PROGRAM Pellet_Calibration
VAR
	SET_CALIBRATON_VALUE : BOOL;

	
	
	Pellet_Length_Temp_Cal_Val : REAL;
END_VAR

 Pellet_Length_Temp_Cal_Val :=  GVL_Pelletizer.Pellet_Length_Inch_Input/ GVL_Pelletizer.Pellet_Length_Measured_Input;


IF SET_CALIBRATON_VALUE THEN
	GVL_Pelletizer.Pellet_Length_Calibration_Value := Pellet_Length_Temp_Cal_Val;
END_IF

END_PROGRAM

(* stored: Version 1.1.0.1, ProductVersion 3.1.4024.12
   POU Pellet_Calibration: Id {237dd450-47a8-4a46-9fe2-c44f1dca051f}, SpecialFunc None *)
